(* Schneider Machine Expert - Basic project Lark_Sobti_Lubrication_TM100, file version 2.2.0.0 *)
(* ProjectInformations: Name=New project *)

HARDWARE
  Cpu 0: TM100C24RN
  EthernetConfiguration: NetworkName=M221, IpAllocationMode=FixedAddress, IpAddress=0.0.0.0, SubnetMask=0.0.0.0
  SerialLineConfiguration: Baud=Baud19200, Parity=ParityEven, DataBits=DataBits8, StopBits=StopBits1, PhysicalMedium=PhysicalMediumRs485, TransmissionMode=TransmissionModeModbusRtu, SlaveId=1, Addressing=SlaveAddressing
  MastTask: UsePeriodScanMode=false, PeriodScan=100
  FastTask: Period=255
  CpuBehavior: StartingMode=StartAsPreviousState, AutoSaveRamOnEeprom=true, WatchdogPeriod=250

SYMBOLS  (address, symbol, comment, settings)
  %M0       AUTOSS
  %M1       LINE2ON1
  %M2       LINE1FBHMI
  %M3       LINE2FBHMI
  %M4       MOTORONHMI
  %M5       MOTORTRIPHMI
  %M6       TANKEMPTYHMI
  %M7       LINE1ON1
  %M8       LINE1REPEAT
  %M9       LINE1ONELAPSED
  %M10      LINE2REPEAT
  %M11      LINE2ONELAPSED
  %M12      STARTCMD
  %M13      LINE1REP1
  %M14      LINE2REP1
  %M16      LINE1ONHMI
  %M17      LINE2ONHMI
  %MW10     LINE1INTTIMEACTHMI
  %MW11     LINE1SETTIMEACTHMI
  %MW12     LINE2INTTIMEACTHMI
  %MW13     LINE2SETTIMEACTHMI
  %MW14     LINE1SETTIMEHMI
  %MW15     LINE1INTTIMEHMI
  %MW16     LINE2SETTIMEHMI
  %MW17     LINE2INTTIMEHMI
  %TM0        [Base=OneSecond, IsRetentive=true]
  %TM1        [IsRetentive=true]
  %TM2        [Base=OneSecond, IsRetentive=true]
  %TM3        [IsRetentive=true]
  %I0.0     MOTORTRIP
  %I0.1     MOTORFB
  %I0.2     MANUALSTART
  %I0.3     MANUALSTOP
  %I0.4     MANUALSS
  %I0.5     LINE2SS
  %I0.6     TANKEMPTY
  %I0.7     SENSOR1
  %I0.8     SENSOR2
  %Q0.0     MOTORCMD
  %Q0.1     VALVECMD

POU New POU
  (* SectionNumber=1 *)

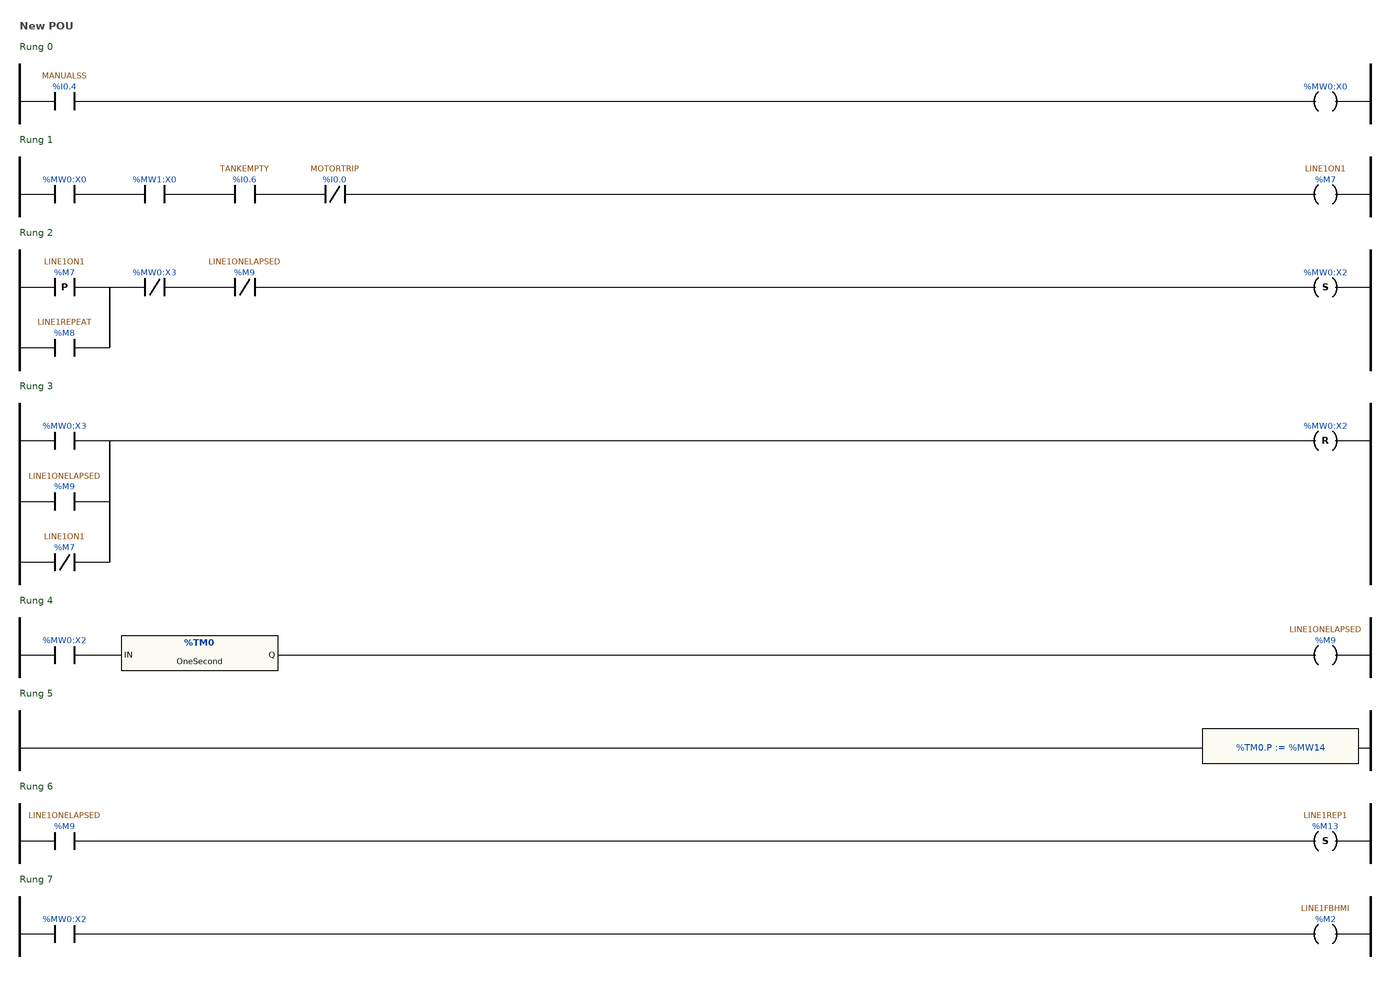

// Rung 0
  LD %I0.4                (* MANUALSS *)
  ST %MW0:X0
  // as ST:
  //   %MW0:X0 := MANUALSS;

// Rung 1
  LD %MW0:X0
  AND %MW1:X0
  AND %I0.6               (* TANKEMPTY *)
  ANDN %I0.0              (* MOTORTRIP *)
  ST %M7                  (* LINE1ON1 *)
  // as ST:
  //   LINE1ON1 := %MW0:X0 AND %MW1:X0 AND TANKEMPTY AND NOT MOTORTRIP;

// Rung 2
  LDR %M7                 (* LINE1ON1 *)
  OR %M8                  (* LINE1REPEAT *)
  ANDN %MW0:X3
  ANDN %M9                (* LINE1ONELAPSED *)
  S %MW0:X2
  // as ST:
  //   IF (RISING(LINE1ON1) OR LINE1REPEAT) AND NOT %MW0:X3 AND NOT LINE1ONELAPSED THEN %MW0:X2 := TRUE; END_IF;

// Rung 3
  LD %MW0:X3
  OR %M9                  (* LINE1ONELAPSED *)
  ORN %M7                 (* LINE1ON1 *)
  R %MW0:X2
  // as ST:
  //   IF %MW0:X3 OR LINE1ONELAPSED OR NOT LINE1ON1 THEN %MW0:X2 := FALSE; END_IF;

// Rung 4
  BLK %TM0
  LD %MW0:X2
  IN
  OUT_BLK
  LD Q
  ST %M9                  (* LINE1ONELAPSED *)
  END_BLK
  // as ST:
  //   %TM0(IN := %MW0:X2);
  //   LINE1ONELAPSED := %TM0.Q;

// Rung 5
  LD 1
  [ %TM0.P := %MW14 ]     (* LINE1SETTIMEHMI *)
  // as ST:
  //   %TM0.P := LINE1SETTIMEHMI;

// Rung 6
  LD %M9                  (* LINE1ONELAPSED *)
  S %M13                  (* LINE1REP1 *)
  // as ST:
  //   IF LINE1ONELAPSED THEN LINE1REP1 := TRUE; END_IF;

// Rung 7
  LD %MW0:X2
  ST %M2                  (* LINE1FBHMI *)
  // as ST:
  //   LINE1FBHMI := %MW0:X2;

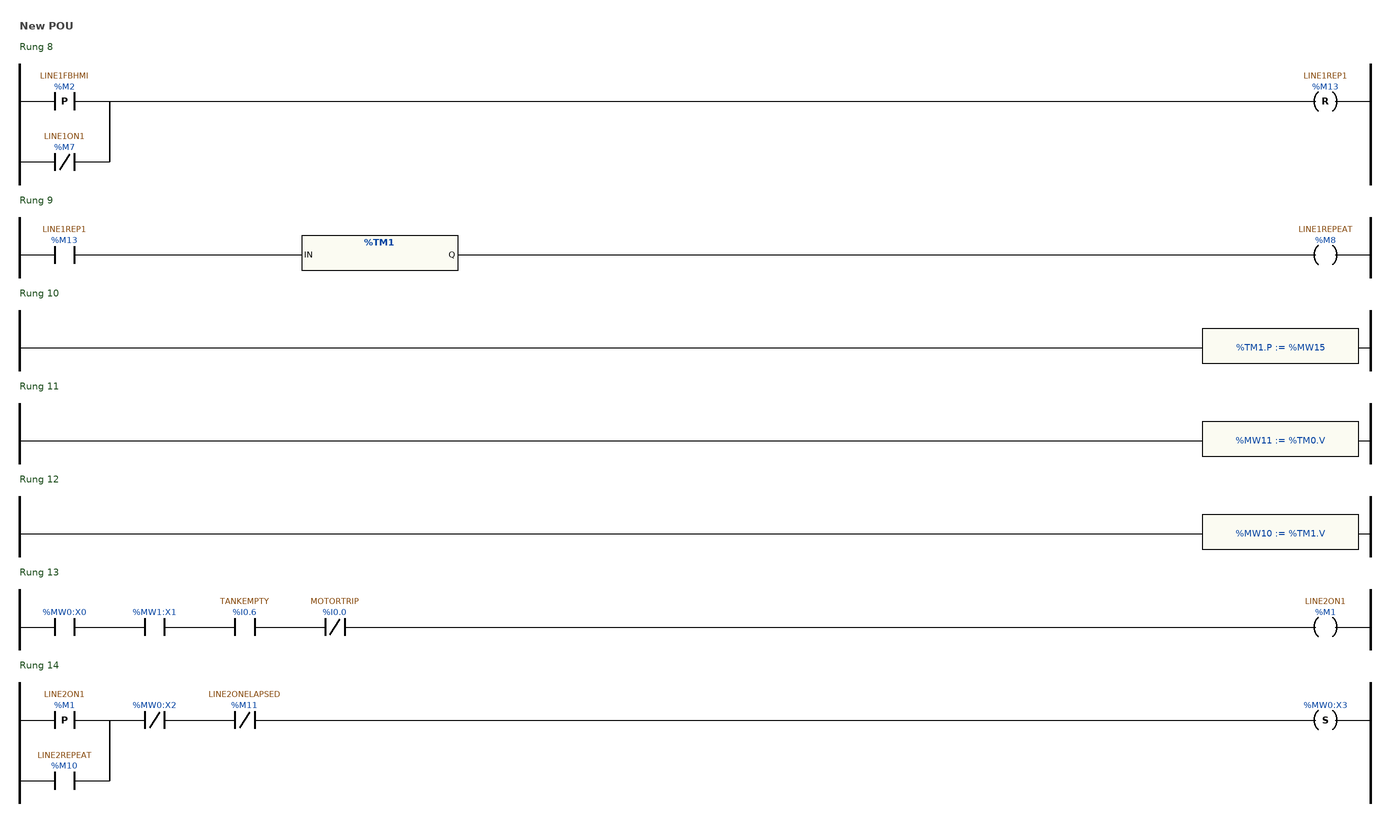

// Rung 8
  LDR %M2                 (* LINE1FBHMI *)
  ORN %M7                 (* LINE1ON1 *)
  R %M13                  (* LINE1REP1 *)
  // as ST:
  //   IF RISING(LINE1FBHMI) OR NOT LINE1ON1 THEN LINE1REP1 := FALSE; END_IF;

// Rung 9
  BLK %TM1
  LD %M13                 (* LINE1REP1 *)
  IN
  OUT_BLK
  LD Q
  ST %M8                  (* LINE1REPEAT *)
  END_BLK
  // as ST:
  //   %TM1(IN := LINE1REP1);
  //   LINE1REPEAT := %TM1.Q;

// Rung 10
  LD 1
  [ %TM1.P := %MW15 ]     (* LINE1INTTIMEHMI *)
  // as ST:
  //   %TM1.P := LINE1INTTIMEHMI;

// Rung 11
  LD 1
  [ %MW11 := %TM0.V ]     (* LINE1SETTIMEACTHMI *)
  // as ST:
  //   LINE1SETTIMEACTHMI := %TM0.V;

// Rung 12
  LD 1
  [ %MW10 := %TM1.V ]     (* LINE1INTTIMEACTHMI *)
  // as ST:
  //   LINE1INTTIMEACTHMI := %TM1.V;

// Rung 13
  LD %MW0:X0
  AND %MW1:X1
  AND %I0.6               (* TANKEMPTY *)
  ANDN %I0.0              (* MOTORTRIP *)
  ST %M1                  (* LINE2ON1 *)
  // as ST:
  //   LINE2ON1 := %MW0:X0 AND %MW1:X1 AND TANKEMPTY AND NOT MOTORTRIP;

// Rung 14
  LDR %M1                 (* LINE2ON1 *)
  OR %M10                 (* LINE2REPEAT *)
  ANDN %MW0:X2
  ANDN %M11               (* LINE2ONELAPSED *)
  S %MW0:X3
  // as ST:
  //   IF (RISING(LINE2ON1) OR LINE2REPEAT) AND NOT %MW0:X2 AND NOT LINE2ONELAPSED THEN %MW0:X3 := TRUE; END_IF;

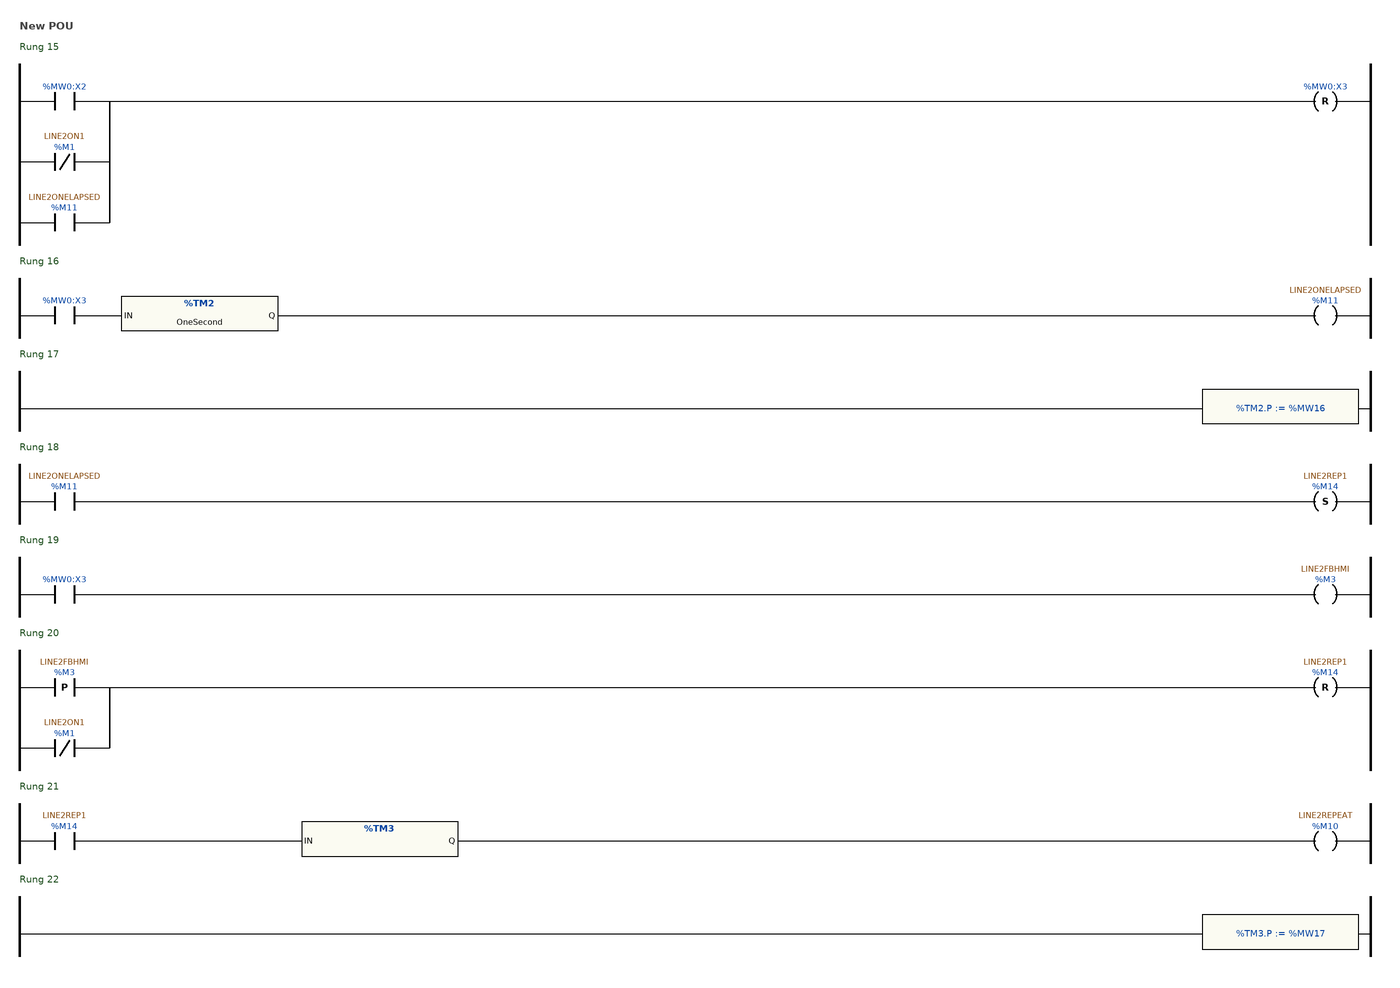

// Rung 15
  LD %MW0:X2
  ORN %M1                 (* LINE2ON1 *)
  OR %M11                 (* LINE2ONELAPSED *)
  R %MW0:X3
  // as ST:
  //   IF %MW0:X2 OR NOT LINE2ON1 OR LINE2ONELAPSED THEN %MW0:X3 := FALSE; END_IF;

// Rung 16
  BLK %TM2
  LD %MW0:X3
  IN
  OUT_BLK
  LD Q
  ST %M11                 (* LINE2ONELAPSED *)
  END_BLK
  // as ST:
  //   %TM2(IN := %MW0:X3);
  //   LINE2ONELAPSED := %TM2.Q;

// Rung 17
  LD 1
  [ %TM2.P := %MW16 ]     (* LINE2SETTIMEHMI *)
  // as ST:
  //   %TM2.P := LINE2SETTIMEHMI;

// Rung 18
  LD %M11                 (* LINE2ONELAPSED *)
  S %M14                  (* LINE2REP1 *)
  // as ST:
  //   IF LINE2ONELAPSED THEN LINE2REP1 := TRUE; END_IF;

// Rung 19
  LD %MW0:X3
  ST %M3                  (* LINE2FBHMI *)
  // as ST:
  //   LINE2FBHMI := %MW0:X3;

// Rung 20
  LDR %M3                 (* LINE2FBHMI *)
  ORN %M1                 (* LINE2ON1 *)
  R %M14                  (* LINE2REP1 *)
  // as ST:
  //   IF RISING(LINE2FBHMI) OR NOT LINE2ON1 THEN LINE2REP1 := FALSE; END_IF;

// Rung 21
  BLK %TM3
  LD %M14                 (* LINE2REP1 *)
  IN
  OUT_BLK
  LD Q
  ST %M10                 (* LINE2REPEAT *)
  END_BLK
  // as ST:
  //   %TM3(IN := LINE2REP1);
  //   LINE2REPEAT := %TM3.Q;

// Rung 22
  LD 1
  [ %TM3.P := %MW17 ]     (* LINE2INTTIMEHMI *)
  // as ST:
  //   %TM3.P := LINE2INTTIMEHMI;

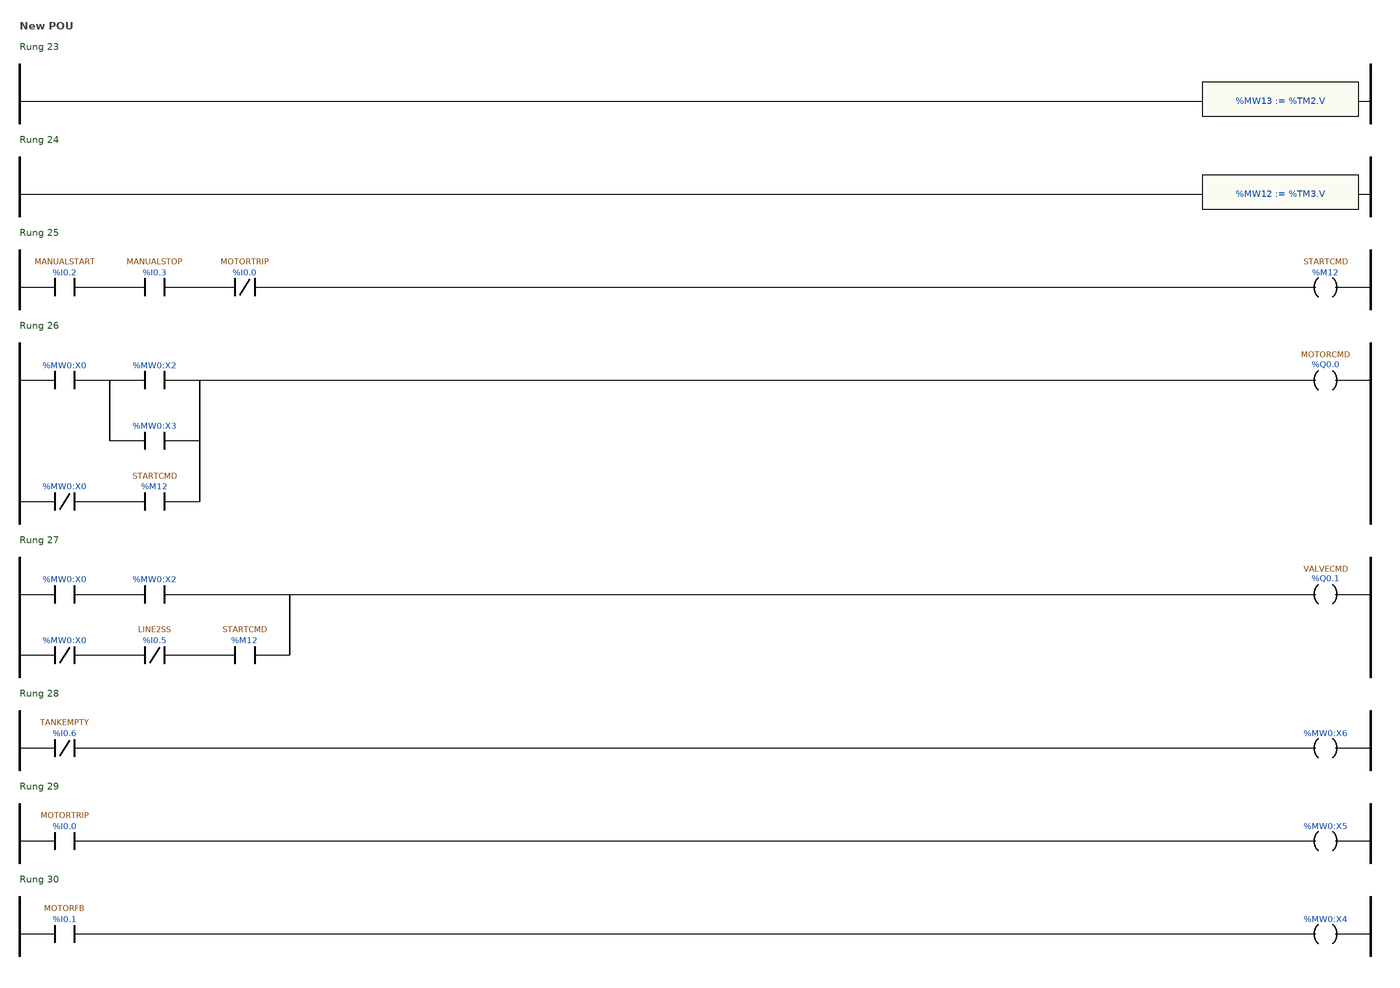

// Rung 23
  LD 1
  [ %MW13 := %TM2.V ]     (* LINE2SETTIMEACTHMI *)
  // as ST:
  //   LINE2SETTIMEACTHMI := %TM2.V;

// Rung 24
  LD 1
  [ %MW12 := %TM3.V ]     (* LINE2INTTIMEACTHMI *)
  // as ST:
  //   LINE2INTTIMEACTHMI := %TM3.V;

// Rung 25
  LD %I0.2                (* MANUALSTART *)
  AND %I0.3               (* MANUALSTOP *)
  ANDN %I0.0              (* MOTORTRIP *)
  ST %M12                 (* STARTCMD *)
  // as ST:
  //   STARTCMD := MANUALSTART AND MANUALSTOP AND NOT MOTORTRIP;

// Rung 26
  LD %MW0:X0
  AND( %MW0:X2
  OR %MW0:X3
  )
  OR(N %MW0:X0
  AND %M12                (* STARTCMD *)
  )
  ST %Q0.0                (* MOTORCMD *)
  // as ST:
  //   MOTORCMD := %MW0:X0 AND (%MW0:X2 OR %MW0:X3) OR NOT %MW0:X0 AND STARTCMD;

// Rung 27
  LD %MW0:X0
  AND %MW0:X2
  OR(N %MW0:X0
  ANDN %I0.5              (* LINE2SS *)
  AND %M12                (* STARTCMD *)
  )
  ST %Q0.1                (* VALVECMD *)
  // as ST:
  //   VALVECMD := %MW0:X0 AND %MW0:X2 OR NOT %MW0:X0 AND NOT LINE2SS AND STARTCMD;

// Rung 28
  LDN %I0.6               (* TANKEMPTY *)
  ST %MW0:X6
  // as ST:
  //   %MW0:X6 := NOT TANKEMPTY;

// Rung 29
  LD %I0.0                (* MOTORTRIP *)
  ST %MW0:X5
  // as ST:
  //   %MW0:X5 := MOTORTRIP;

// Rung 30
  LD %I0.1                (* MOTORFB *)
  ST %MW0:X4
  // as ST:
  //   %MW0:X4 := MOTORFB;
